// TwinCAT 3 PLC project TestIOC
// ProgramVersion: 3.1.4026.17
// libraries:
//   LCLS General, * (SLAC)
//   LCLS Vacuum, * (SLAC - LCLS)
//   lcls-twincat-common-components, * (SLAC)
//   lcls-twincat-math, * (SLAC - LCLS)
//   lcls-twincat-motion, * (SLAC)
//   lcls-twincat-optics, * (SLAC)
//   lcls-twincat-physics, * (SLAC)
//   LCLS_MotionAbstraction, * (SLAC)
//   LCLS_Tc_DevAbs, * (SLAC - LCLS)
//   PMPS, * (SLAC - LCLS)
//   Tc2_MC2, * (Beckhoff Automation GmbH)
//   Tc2_Standard, * (Beckhoff Automation GmbH)
//   Tc2_System, * (Beckhoff Automation GmbH)
//   Tc3_Module, * (Beckhoff Automation GmbH)
//   TcUnit, * (www.tcunit.org)
// project tree:
//   DUTs/ ENUM_Test.TcDUT, ST_NestedTypes01.TcDUT, ST_NestedTypes02.TcDUT, ST_NestedTypes03.TcDUT, ST_NestedTypes04.TcDUT, ST_NestedTypes05.TcDUT, ST_PytmcTypes.TcDUT
//   GVLs/ GVL.TcGVL
//   / PlcTask.TcTTO
//   POUs/ Main.TcPOU, F_UpdateArray.TcPOU
// real-time tasks:
//   TASK PlcTask: cycle T#10ms, priority 20, ADS port 350
// motion (NC):
//   TASK NC-Task 1 SAF: cycle T#2ms, priority 4, ADS port 501
//   TASK NC-Task 1 SVB: cycle T#10ms, priority 8, ADS port 511
//   AXIS Axis 1 (id 1)
//     OtherSettings: AllowMotionCmdToSlave=true
//     encoder EncType=1
//     drive DrvType=5
//       Analog: TorqueSetpointScale=10, ScaleFactorActTorque=0.1
//       TimeComp: TaskDelayCycles=1
//     controller CtrType=1
//       CtrPara: PriorControlFactor=1
//         Observer: BandWidth=20
//   AXIS Axis 2 (id 2)
//     OtherSettings: AllowMotionCmdToSlave=true
//     encoder EncType=1
//     drive DrvType=5
//       Analog: TorqueSetpointScale=10, ScaleFactorActTorque=0.1
//       TimeComp: TaskDelayCycles=1
//     controller CtrType=1
//       CtrPara: PriorControlFactor=1
//         Observer: BandWidth=20
//   AXIS Axis 3 (id 3)
//     OtherSettings: AllowMotionCmdToSlave=true
//     encoder EncType=1
//     drive DrvType=5
//       Analog: TorqueSetpointScale=10, ScaleFactorActTorque=0.1
//       TimeComp: TaskDelayCycles=1
//     controller CtrType=1
//       CtrPara: PriorControlFactor=1
//         Observer: BandWidth=20
//   AXIS Axis 4 (id 4)
//     OtherSettings: AllowMotionCmdToSlave=true
//     encoder EncType=1
//     drive DrvType=5
//       Analog: TorqueSetpointScale=10, ScaleFactorActTorque=0.1
//       TimeComp: TaskDelayCycles=1
//     controller CtrType=1
//       CtrPara: PriorControlFactor=1
//         Observer: BandWidth=20
//   AXIS Axis 5 (id 5)
//     OtherSettings: AllowMotionCmdToSlave=true
//     encoder EncType=1
//     drive DrvType=5
//       Analog: TorqueSetpointScale=10, ScaleFactorActTorque=0.1
//       TimeComp: TaskDelayCycles=1
//     controller CtrType=1
//       CtrPara: PriorControlFactor=1
//         Observer: BandWidth=20
//   AXIS Axis 6 (id 6)
//     OtherSettings: AllowMotionCmdToSlave=true
//     encoder EncType=1
//     drive DrvType=5
//       Analog: TorqueSetpointScale=10, ScaleFactorActTorque=0.1
//       TimeComp: TaskDelayCycles=1
//     controller CtrType=1
//       CtrPara: PriorControlFactor=1
//         Observer: BandWidth=20
//   AXIS Axis 7 (id 7)
//     OtherSettings: AllowMotionCmdToSlave=true
//     encoder EncType=1
//     drive DrvType=5
//       Analog: TorqueSetpointScale=10, ScaleFactorActTorque=0.1
//       TimeComp: TaskDelayCycles=1
//     controller CtrType=1
//       CtrPara: PriorControlFactor=1
//         Observer: BandWidth=20
//   AXIS Axis 8 (id 8)
//     OtherSettings: AllowMotionCmdToSlave=true
//     encoder EncType=1
//     drive DrvType=5
//       Analog: TorqueSetpointScale=10, ScaleFactorActTorque=0.1
//       TimeComp: TaskDelayCycles=1
//     controller CtrType=1
//       CtrPara: PriorControlFactor=1
//         Observer: BandWidth=20
//   AXIS Axis 9 (id 9)
//     OtherSettings: AllowMotionCmdToSlave=true
//     encoder EncType=1
//     drive DrvType=5
//       Analog: TorqueSetpointScale=10, ScaleFactorActTorque=0.1
//       TimeComp: TaskDelayCycles=1
//     controller CtrType=1
//       CtrPara: PriorControlFactor=1
//         Observer: BandWidth=20
//   AXIS Axis 10 (id 10)
//     OtherSettings: AllowMotionCmdToSlave=true
//     encoder EncType=1
//     drive DrvType=5
//       Analog: TorqueSetpointScale=10, ScaleFactorActTorque=0.1
//       TimeComp: TaskDelayCycles=1
//     controller CtrType=1
//       CtrPara: PriorControlFactor=1
//         Observer: BandWidth=20
//   AXIS Axis 11 (id 11)
//     OtherSettings: AllowMotionCmdToSlave=true
//     encoder EncType=1
//     drive DrvType=5
//       Analog: TorqueSetpointScale=10, ScaleFactorActTorque=0.1
//       TimeComp: TaskDelayCycles=1
//     controller CtrType=1
//       CtrPara: PriorControlFactor=1
//         Observer: BandWidth=20
//   AXIS Axis 12 (id 12)
//     OtherSettings: AllowMotionCmdToSlave=true
//     encoder EncType=1
//     drive DrvType=5
//       Analog: TorqueSetpointScale=10, ScaleFactorActTorque=0.1
//       TimeComp: TaskDelayCycles=1
//     controller CtrType=1
//       CtrPara: PriorControlFactor=1
//         Observer: BandWidth=20
//   AXIS Axis 13 (id 13)
//     OtherSettings: AllowMotionCmdToSlave=true
//     encoder EncType=1
//     drive DrvType=5
//       Analog: TorqueSetpointScale=10, ScaleFactorActTorque=0.1
//       TimeComp: TaskDelayCycles=1
//     controller CtrType=1
//       CtrPara: PriorControlFactor=1
//         Observer: BandWidth=20
//   AXIS Axis 14 (id 14)
//     OtherSettings: AllowMotionCmdToSlave=true
//     encoder EncType=1
//     drive DrvType=5
//       Analog: TorqueSetpointScale=10, ScaleFactorActTorque=0.1
//       TimeComp: TaskDelayCycles=1
//     controller CtrType=1
//       CtrPara: PriorControlFactor=1
//         Observer: BandWidth=20
//   AXIS Axis 15 (id 15)
//     OtherSettings: AllowMotionCmdToSlave=true
//     encoder EncType=1
//     drive DrvType=5
//       Analog: TorqueSetpointScale=10, ScaleFactorActTorque=0.1
//       TimeComp: TaskDelayCycles=1
//     controller CtrType=1
//       CtrPara: PriorControlFactor=1
//         Observer: BandWidth=20
//   AXIS Axis 16 (id 16)
//     OtherSettings: AllowMotionCmdToSlave=true
//     encoder EncType=1
//     drive DrvType=5
//       Analog: TorqueSetpointScale=10, ScaleFactorActTorque=0.1
//       TimeComp: TaskDelayCycles=1
//     controller CtrType=1
//       CtrPara: PriorControlFactor=1
//         Observer: BandWidth=20
//   AXIS Axis 17 (id 17)
//     OtherSettings: AllowMotionCmdToSlave=true
//     encoder EncType=1
//     drive DrvType=5
//       Analog: TorqueSetpointScale=10, ScaleFactorActTorque=0.1
//       TimeComp: TaskDelayCycles=1
//     controller CtrType=1
//       CtrPara: PriorControlFactor=1
//         Observer: BandWidth=20
//   AXIS Axis 18 (id 18)
//     OtherSettings: AllowMotionCmdToSlave=true
//     encoder EncType=1
//     drive DrvType=5
//       Analog: TorqueSetpointScale=10, ScaleFactorActTorque=0.1
//       TimeComp: TaskDelayCycles=1
//     controller CtrType=1
//       CtrPara: PriorControlFactor=1
//         Observer: BandWidth=20
//   AXIS Axis 19 (id 19)
//     OtherSettings: AllowMotionCmdToSlave=true
//     encoder EncType=1
//     drive DrvType=5
//       Analog: TorqueSetpointScale=10, ScaleFactorActTorque=0.1
//       TimeComp: TaskDelayCycles=1
//     controller CtrType=1
//       CtrPara: PriorControlFactor=1
//         Observer: BandWidth=20
//   AXIS Axis 20 (id 20)
//     OtherSettings: AllowMotionCmdToSlave=true
//     encoder EncType=1
//     drive DrvType=5
//       Analog: TorqueSetpointScale=10, ScaleFactorActTorque=0.1
//       TimeComp: TaskDelayCycles=1
//     controller CtrType=1
//       CtrPara: PriorControlFactor=1
//         Observer: BandWidth=20
//   AXIS Axis 21 (id 21)
//     OtherSettings: AllowMotionCmdToSlave=true
//     encoder EncType=1
//     drive DrvType=5
//       Analog: TorqueSetpointScale=10, ScaleFactorActTorque=0.1
//       TimeComp: TaskDelayCycles=1
//     controller CtrType=1
//       CtrPara: PriorControlFactor=1
//         Observer: BandWidth=20
//   AXIS Axis 22 (id 22)
//     OtherSettings: AllowMotionCmdToSlave=true
//     encoder EncType=1
//     drive DrvType=5
//       Analog: TorqueSetpointScale=10, ScaleFactorActTorque=0.1
//       TimeComp: TaskDelayCycles=1
//     controller CtrType=1
//       CtrPara: PriorControlFactor=1
//         Observer: BandWidth=20
//   AXIS Axis 23 (id 23)
//     OtherSettings: AllowMotionCmdToSlave=true
//     encoder EncType=1
//     drive DrvType=5
//       Analog: TorqueSetpointScale=10, ScaleFactorActTorque=0.1
//       TimeComp: TaskDelayCycles=1
//     controller CtrType=1
//       CtrPara: PriorControlFactor=1
//         Observer: BandWidth=20
//   AXIS Axis 24 (id 24)
//     OtherSettings: AllowMotionCmdToSlave=true
//     encoder EncType=1
//     drive DrvType=5
//       Analog: TorqueSetpointScale=10, ScaleFactorActTorque=0.1
//       TimeComp: TaskDelayCycles=1
//     controller CtrType=1
//       CtrPara: PriorControlFactor=1
//         Observer: BandWidth=20
//   AXIS Axis 25 (id 25)
//     OtherSettings: AllowMotionCmdToSlave=true
//     encoder EncType=1
//     drive DrvType=5
//       Analog: TorqueSetpointScale=10, ScaleFactorActTorque=0.1
//       TimeComp: TaskDelayCycles=1
//     controller CtrType=1
//       CtrPara: PriorControlFactor=1
//         Observer: BandWidth=20
//   AXIS Axis 26 (id 26)
//     OtherSettings: AllowMotionCmdToSlave=true
//     encoder EncType=1
//     drive DrvType=5
//       Analog: TorqueSetpointScale=10, ScaleFactorActTorque=0.1
//       TimeComp: TaskDelayCycles=1
//     controller CtrType=1
//       CtrPara: PriorControlFactor=1
//         Observer: BandWidth=20
//   AXIS Axis 27 (id 27)
//     OtherSettings: AllowMotionCmdToSlave=true
//     encoder EncType=1
//     drive DrvType=5
//       Analog: TorqueSetpointScale=10, ScaleFactorActTorque=0.1
//       TimeComp: TaskDelayCycles=1
//     controller CtrType=1
//       CtrPara: PriorControlFactor=1
//         Observer: BandWidth=20
//   AXIS Axis 28 (id 28)
//     OtherSettings: AllowMotionCmdToSlave=true
//     encoder EncType=1
//     drive DrvType=5
//       Analog: TorqueSetpointScale=10, ScaleFactorActTorque=0.1
//       TimeComp: TaskDelayCycles=1
//     controller CtrType=1
//       CtrPara: PriorControlFactor=1
//         Observer: BandWidth=20
//   AXIS Axis 29 (id 29)
//     OtherSettings: AllowMotionCmdToSlave=true
//     encoder EncType=1
//     drive DrvType=5
//       Analog: TorqueSetpointScale=10, ScaleFactorActTorque=0.1
//       TimeComp: TaskDelayCycles=1
//     controller CtrType=1
//       CtrPara: PriorControlFactor=1
//         Observer: BandWidth=20
//   AXIS Axis 30 (id 30)
//     OtherSettings: AllowMotionCmdToSlave=true
//     encoder EncType=1
//     drive DrvType=5
//       Analog: TorqueSetpointScale=10, ScaleFactorActTorque=0.1
//       TimeComp: TaskDelayCycles=1
//     controller CtrType=1
//       CtrPara: PriorControlFactor=1
//         Observer: BandWidth=20
//   AXIS Axis 31 (id 31)
//     OtherSettings: AllowMotionCmdToSlave=true
//     encoder EncType=1
//     drive DrvType=5
//       Analog: TorqueSetpointScale=10, ScaleFactorActTorque=0.1
//       TimeComp: TaskDelayCycles=1
//     controller CtrType=1
//       CtrPara: PriorControlFactor=1
//         Observer: BandWidth=20
//   AXIS Axis 32 (id 32)
//     OtherSettings: AllowMotionCmdToSlave=true
//     encoder EncType=1
//     drive DrvType=5
//       Analog: TorqueSetpointScale=10, ScaleFactorActTorque=0.1
//       TimeComp: TaskDelayCycles=1
//     controller CtrType=1
//       CtrPara: PriorControlFactor=1
//         Observer: BandWidth=20
//   AXIS Axis 33 (id 33)
//     OtherSettings: AllowMotionCmdToSlave=true
//     encoder EncType=1
//     drive DrvType=5
//       Analog: TorqueSetpointScale=10, ScaleFactorActTorque=0.1
//       TimeComp: TaskDelayCycles=1
//     controller CtrType=1
//       CtrPara: PriorControlFactor=1
//         Observer: BandWidth=20
//   AXIS Axis 34 (id 34)
//     OtherSettings: AllowMotionCmdToSlave=true
//     encoder EncType=1
//     drive DrvType=5
//       Analog: TorqueSetpointScale=10, ScaleFactorActTorque=0.1
//       TimeComp: TaskDelayCycles=1
//     controller CtrType=1
//       CtrPara: PriorControlFactor=1
//         Observer: BandWidth=20
//   AXIS Axis 35 (id 35)
//     OtherSettings: AllowMotionCmdToSlave=true
//     encoder EncType=1
//     drive DrvType=5
//       Analog: TorqueSetpointScale=10, ScaleFactorActTorque=0.1
//       TimeComp: TaskDelayCycles=1
//     controller CtrType=1
//       CtrPara: PriorControlFactor=1
//         Observer: BandWidth=20
//   AXIS Axis 36 (id 36)
//     OtherSettings: AllowMotionCmdToSlave=true
//     encoder EncType=1
//     drive DrvType=5
//       Analog: TorqueSetpointScale=10, ScaleFactorActTorque=0.1
//       TimeComp: TaskDelayCycles=1
//     controller CtrType=1
//       CtrPara: PriorControlFactor=1
//         Observer: BandWidth=20
//   AXIS Axis 37 (id 37)
//     OtherSettings: AllowMotionCmdToSlave=true
//     encoder EncType=1
//     drive DrvType=5
//       Analog: TorqueSetpointScale=10, ScaleFactorActTorque=0.1
//       TimeComp: TaskDelayCycles=1
//     controller CtrType=1
//       CtrPara: PriorControlFactor=1
//         Observer: BandWidth=20
//   AXIS Axis 38 (id 38)
//     OtherSettings: AllowMotionCmdToSlave=true
//     encoder EncType=1
//     drive DrvType=5
//       Analog: TorqueSetpointScale=10, ScaleFactorActTorque=0.1
//       TimeComp: TaskDelayCycles=1
//     controller CtrType=1
//       CtrPara: PriorControlFactor=1
//         Observer: BandWidth=20
//   AXIS Axis 39 (id 39)
//     OtherSettings: AllowMotionCmdToSlave=true
//     encoder EncType=1
//     drive DrvType=5
//       Analog: TorqueSetpointScale=10, ScaleFactorActTorque=0.1
//       TimeComp: TaskDelayCycles=1
//     controller CtrType=1
//       CtrPara: PriorControlFactor=1
//         Observer: BandWidth=20
//   AXIS Axis 40 (id 40)
//     OtherSettings: AllowMotionCmdToSlave=true
//     encoder EncType=1
//     drive DrvType=5
//       Analog: TorqueSetpointScale=10, ScaleFactorActTorque=0.1
//       TimeComp: TaskDelayCycles=1
//     controller CtrType=1
//       CtrPara: PriorControlFactor=1
//         Observer: BandWidth=20
//   AXIS Axis 41 (id 41)
//     OtherSettings: AllowMotionCmdToSlave=true
//     encoder EncType=1
//     drive DrvType=5
//       Analog: TorqueSetpointScale=10, ScaleFactorActTorque=0.1
//       TimeComp: TaskDelayCycles=1
//     controller CtrType=1
//       CtrPara: PriorControlFactor=1
//         Observer: BandWidth=20
//   AXIS Axis 42 (id 42)
//     OtherSettings: AllowMotionCmdToSlave=true
//     encoder EncType=1
//     drive DrvType=5
//       Analog: TorqueSetpointScale=10, ScaleFactorActTorque=0.1
//       TimeComp: TaskDelayCycles=1
//     controller CtrType=1
//       CtrPara: PriorControlFactor=1
//         Observer: BandWidth=20
//   AXIS Axis 43 (id 43)
//     OtherSettings: AllowMotionCmdToSlave=true
//     encoder EncType=1
//     drive DrvType=5
//       Analog: TorqueSetpointScale=10, ScaleFactorActTorque=0.1
//       TimeComp: TaskDelayCycles=1
//     controller CtrType=1
//       CtrPara: PriorControlFactor=1
//         Observer: BandWidth=20
//   AXIS Axis 44 (id 44)
//     OtherSettings: AllowMotionCmdToSlave=true
//     encoder EncType=1
//     drive DrvType=5
//       Analog: TorqueSetpointScale=10, ScaleFactorActTorque=0.1
//       TimeComp: TaskDelayCycles=1
//     controller CtrType=1
//       CtrPara: PriorControlFactor=1
//         Observer: BandWidth=20
//   AXIS Axis 45 (id 45)
//     OtherSettings: AllowMotionCmdToSlave=true
//     encoder EncType=1
//     drive DrvType=5
//       Analog: TorqueSetpointScale=10, ScaleFactorActTorque=0.1
//       TimeComp: TaskDelayCycles=1
//     controller CtrType=1
//       CtrPara: PriorControlFactor=1
//         Observer: BandWidth=20
//   AXIS Axis 46 (id 46)
//     OtherSettings: AllowMotionCmdToSlave=true
//     encoder EncType=1
//     drive DrvType=5
//       Analog: TorqueSetpointScale=10, ScaleFactorActTorque=0.1
//       TimeComp: TaskDelayCycles=1
//     controller CtrType=1
//       CtrPara: PriorControlFactor=1
//         Observer: BandWidth=20
//   AXIS Axis 47 (id 47)
//     OtherSettings: AllowMotionCmdToSlave=true
//     encoder EncType=1
//     drive DrvType=5
//       Analog: TorqueSetpointScale=10, ScaleFactorActTorque=0.1
//       TimeComp: TaskDelayCycles=1
//     controller CtrType=1
//       CtrPara: PriorControlFactor=1
//         Observer: BandWidth=20
//   AXIS Axis 48 (id 48)
//     OtherSettings: AllowMotionCmdToSlave=true
//     encoder EncType=1
//     drive DrvType=5
//       Analog: TorqueSetpointScale=10, ScaleFactorActTorque=0.1
//       TimeComp: TaskDelayCycles=1
//     controller CtrType=1
//       CtrPara: PriorControlFactor=1
//         Observer: BandWidth=20
//   AXIS Axis 49 (id 49)
//     OtherSettings: AllowMotionCmdToSlave=true
//     encoder EncType=1
//     drive DrvType=5
//       Analog: TorqueSetpointScale=10, ScaleFactorActTorque=0.1
//       TimeComp: TaskDelayCycles=1
//     controller CtrType=1
//       CtrPara: PriorControlFactor=1
//         Observer: BandWidth=20
//   AXIS Axis 50 (id 50)
//     OtherSettings: AllowMotionCmdToSlave=true
//     encoder EncType=1
//     drive DrvType=5
//       Analog: TorqueSetpointScale=10, ScaleFactorActTorque=0.1
//       TimeComp: TaskDelayCycles=1
//     controller CtrType=1
//       CtrPara: PriorControlFactor=1
//         Observer: BandWidth=20
//   AXIS Axis 51 (id 51)
//     OtherSettings: AllowMotionCmdToSlave=true
//     encoder EncType=1
//     drive DrvType=5
//       Analog: TorqueSetpointScale=10, ScaleFactorActTorque=0.1
//       TimeComp: TaskDelayCycles=1
//     controller CtrType=1
//       CtrPara: PriorControlFactor=1
//         Observer: BandWidth=20
//   AXIS Axis 52 (id 52)
//     OtherSettings: AllowMotionCmdToSlave=true
//     encoder EncType=1
//     drive DrvType=5
//       Analog: TorqueSetpointScale=10, ScaleFactorActTorque=0.1
//       TimeComp: TaskDelayCycles=1
//     controller CtrType=1
//       CtrPara: PriorControlFactor=1
//         Observer: BandWidth=20
// variable links:
//   (this object) <-> NC-Task 1 SAF/Axes/Axis 1
//     PlcTask Inputs/Main.M1.Axis.NcToPlc <-> Outputs/ToPlc
//     PlcTask Outputs/Main.M1.Axis.PlcToNc <-> Inputs/FromPlc
//   (this object) <-> NC-Task 1 SAF/Axes/Axis 10
//     PlcTask Inputs/Main.aAxisRef[8].NcToPlc <-> Outputs/ToPlc
//     PlcTask Outputs/Main.aAxisRef[8].PlcToNc <-> Inputs/FromPlc
//   (this object) <-> NC-Task 1 SAF/Axes/Axis 11
//     PlcTask Inputs/Main.aAxisRef[9].NcToPlc <-> Outputs/ToPlc
//     PlcTask Outputs/Main.aAxisRef[9].PlcToNc <-> Inputs/FromPlc
//   (this object) <-> NC-Task 1 SAF/Axes/Axis 12
//     PlcTask Inputs/Main.aAxisRef[10].NcToPlc <-> Outputs/ToPlc
//     PlcTask Outputs/Main.aAxisRef[10].PlcToNc <-> Inputs/FromPlc
//   (this object) <-> NC-Task 1 SAF/Axes/Axis 13
//     PlcTask Inputs/Main.aAxisRef[11].NcToPlc <-> Outputs/ToPlc
//     PlcTask Outputs/Main.aAxisRef[11].PlcToNc <-> Inputs/FromPlc
//   (this object) <-> NC-Task 1 SAF/Axes/Axis 14
//     PlcTask Inputs/Main.aAxisRef[12].NcToPlc <-> Outputs/ToPlc
//     PlcTask Outputs/Main.aAxisRef[12].PlcToNc <-> Inputs/FromPlc
//   (this object) <-> NC-Task 1 SAF/Axes/Axis 15
//     PlcTask Inputs/Main.aAxisRef[13].NcToPlc <-> Outputs/ToPlc
//     PlcTask Outputs/Main.aAxisRef[13].PlcToNc <-> Inputs/FromPlc
//   (this object) <-> NC-Task 1 SAF/Axes/Axis 16
//     PlcTask Inputs/Main.aAxisRef[14].NcToPlc <-> Outputs/ToPlc
//     PlcTask Outputs/Main.aAxisRef[14].PlcToNc <-> Inputs/FromPlc
//   (this object) <-> NC-Task 1 SAF/Axes/Axis 17
//     PlcTask Inputs/Main.aAxisRef[15].NcToPlc <-> Outputs/ToPlc
//     PlcTask Outputs/Main.aAxisRef[15].PlcToNc <-> Inputs/FromPlc
//   (this object) <-> NC-Task 1 SAF/Axes/Axis 18
//     PlcTask Inputs/Main.aAxisRef[16].NcToPlc <-> Outputs/ToPlc
//     PlcTask Outputs/Main.aAxisRef[16].PlcToNc <-> Inputs/FromPlc
//   (this object) <-> NC-Task 1 SAF/Axes/Axis 19
//     PlcTask Inputs/Main.aAxisRef[17].NcToPlc <-> Outputs/ToPlc
//     PlcTask Outputs/Main.aAxisRef[17].PlcToNc <-> Inputs/FromPlc
//   (this object) <-> NC-Task 1 SAF/Axes/Axis 2
//     PlcTask Inputs/Main.M2.Axis.NcToPlc <-> Outputs/ToPlc
//     PlcTask Outputs/Main.M2.Axis.PlcToNc <-> Inputs/FromPlc
//   (this object) <-> NC-Task 1 SAF/Axes/Axis 20
//     PlcTask Inputs/Main.aAxisRef[18].NcToPlc <-> Outputs/ToPlc
//     PlcTask Outputs/Main.aAxisRef[18].PlcToNc <-> Inputs/FromPlc
//   (this object) <-> NC-Task 1 SAF/Axes/Axis 21
//     PlcTask Inputs/Main.aAxisRef[19].NcToPlc <-> Outputs/ToPlc
//     PlcTask Outputs/Main.aAxisRef[19].PlcToNc <-> Inputs/FromPlc
//   (this object) <-> NC-Task 1 SAF/Axes/Axis 22
//     PlcTask Inputs/Main.aAxisRef[20].NcToPlc <-> Outputs/ToPlc
//     PlcTask Outputs/Main.aAxisRef[20].PlcToNc <-> Inputs/FromPlc
//   (this object) <-> NC-Task 1 SAF/Axes/Axis 23
//     PlcTask Inputs/Main.aAxisRef[21].NcToPlc <-> Outputs/ToPlc
//     PlcTask Outputs/Main.aAxisRef[21].PlcToNc <-> Inputs/FromPlc
//   (this object) <-> NC-Task 1 SAF/Axes/Axis 24
//     PlcTask Inputs/Main.aAxisRef[22].NcToPlc <-> Outputs/ToPlc
//     PlcTask Outputs/Main.aAxisRef[22].PlcToNc <-> Inputs/FromPlc
//   (this object) <-> NC-Task 1 SAF/Axes/Axis 25
//     PlcTask Inputs/Main.aAxisRef[23].NcToPlc <-> Outputs/ToPlc
//     PlcTask Outputs/Main.aAxisRef[23].PlcToNc <-> Inputs/FromPlc
//   (this object) <-> NC-Task 1 SAF/Axes/Axis 26
//     PlcTask Inputs/Main.aAxisRef[24].NcToPlc <-> Outputs/ToPlc
//     PlcTask Outputs/Main.aAxisRef[24].PlcToNc <-> Inputs/FromPlc
//   (this object) <-> NC-Task 1 SAF/Axes/Axis 27
//     PlcTask Inputs/Main.aAxisRef[25].NcToPlc <-> Outputs/ToPlc
//     PlcTask Outputs/Main.aAxisRef[25].PlcToNc <-> Inputs/FromPlc
//   (this object) <-> NC-Task 1 SAF/Axes/Axis 28
//     PlcTask Inputs/Main.aAxisRef[26].NcToPlc <-> Outputs/ToPlc
//     PlcTask Outputs/Main.aAxisRef[26].PlcToNc <-> Inputs/FromPlc
//   (this object) <-> NC-Task 1 SAF/Axes/Axis 29
//     PlcTask Inputs/Main.aAxisRef[27].NcToPlc <-> Outputs/ToPlc
//     PlcTask Outputs/Main.aAxisRef[27].PlcToNc <-> Inputs/FromPlc
//   (this object) <-> NC-Task 1 SAF/Axes/Axis 3
//     PlcTask Inputs/Main.aAxisRef[1].NcToPlc <-> Outputs/ToPlc
//     PlcTask Outputs/Main.aAxisRef[1].PlcToNc <-> Inputs/FromPlc
//   (this object) <-> NC-Task 1 SAF/Axes/Axis 30
//     PlcTask Inputs/Main.aAxisRef[28].NcToPlc <-> Outputs/ToPlc
//     PlcTask Outputs/Main.aAxisRef[28].PlcToNc <-> Inputs/FromPlc
//   (this object) <-> NC-Task 1 SAF/Axes/Axis 31
//     PlcTask Inputs/Main.aAxisRef[29].NcToPlc <-> Outputs/ToPlc
//     PlcTask Outputs/Main.aAxisRef[29].PlcToNc <-> Inputs/FromPlc
//   (this object) <-> NC-Task 1 SAF/Axes/Axis 32
//     PlcTask Inputs/Main.aAxisRef[30].NcToPlc <-> Outputs/ToPlc
//     PlcTask Outputs/Main.aAxisRef[30].PlcToNc <-> Inputs/FromPlc
//   (this object) <-> NC-Task 1 SAF/Axes/Axis 33
//     PlcTask Inputs/Main.aAxisRef[31].NcToPlc <-> Outputs/ToPlc
//     PlcTask Outputs/Main.aAxisRef[31].PlcToNc <-> Inputs/FromPlc
//   (this object) <-> NC-Task 1 SAF/Axes/Axis 34
//     PlcTask Inputs/Main.aAxisRef[32].NcToPlc <-> Outputs/ToPlc
//     PlcTask Outputs/Main.aAxisRef[32].PlcToNc <-> Inputs/FromPlc
//   (this object) <-> NC-Task 1 SAF/Axes/Axis 35
//     PlcTask Inputs/Main.aAxisRef[33].NcToPlc <-> Outputs/ToPlc
//     PlcTask Outputs/Main.aAxisRef[33].PlcToNc <-> Inputs/FromPlc
//   (this object) <-> NC-Task 1 SAF/Axes/Axis 36
//     PlcTask Inputs/Main.aAxisRef[34].NcToPlc <-> Outputs/ToPlc
//     PlcTask Outputs/Main.aAxisRef[34].PlcToNc <-> Inputs/FromPlc
//   (this object) <-> NC-Task 1 SAF/Axes/Axis 37
//     PlcTask Inputs/Main.aAxisRef[35].NcToPlc <-> Outputs/ToPlc
//     PlcTask Outputs/Main.aAxisRef[35].PlcToNc <-> Inputs/FromPlc
//   (this object) <-> NC-Task 1 SAF/Axes/Axis 38
//     PlcTask Inputs/Main.aAxisRef[36].NcToPlc <-> Outputs/ToPlc
//     PlcTask Outputs/Main.aAxisRef[36].PlcToNc <-> Inputs/FromPlc
//   (this object) <-> NC-Task 1 SAF/Axes/Axis 39
//     PlcTask Inputs/Main.aAxisRef[37].NcToPlc <-> Outputs/ToPlc
//     PlcTask Outputs/Main.aAxisRef[37].PlcToNc <-> Inputs/FromPlc
//   (this object) <-> NC-Task 1 SAF/Axes/Axis 4
//     PlcTask Inputs/Main.aAxisRef[2].NcToPlc <-> Outputs/ToPlc
//     PlcTask Outputs/Main.aAxisRef[2].PlcToNc <-> Inputs/FromPlc
//   (this object) <-> NC-Task 1 SAF/Axes/Axis 40
//     PlcTask Inputs/Main.aAxisRef[38].NcToPlc <-> Outputs/ToPlc
//     PlcTask Outputs/Main.aAxisRef[38].PlcToNc <-> Inputs/FromPlc
//   (this object) <-> NC-Task 1 SAF/Axes/Axis 41
//     PlcTask Inputs/Main.aAxisRef[39].NcToPlc <-> Outputs/ToPlc
//     PlcTask Outputs/Main.aAxisRef[39].PlcToNc <-> Inputs/FromPlc
//   (this object) <-> NC-Task 1 SAF/Axes/Axis 42
//     PlcTask Inputs/Main.aAxisRef[40].NcToPlc <-> Outputs/ToPlc
//     PlcTask Outputs/Main.aAxisRef[40].PlcToNc <-> Inputs/FromPlc
//   (this object) <-> NC-Task 1 SAF/Axes/Axis 43
//     PlcTask Inputs/Main.aAxisRef[41].NcToPlc <-> Outputs/ToPlc
//     PlcTask Outputs/Main.aAxisRef[41].PlcToNc <-> Inputs/FromPlc
//   (this object) <-> NC-Task 1 SAF/Axes/Axis 44
//     PlcTask Inputs/Main.aAxisRef[42].NcToPlc <-> Outputs/ToPlc
//     PlcTask Outputs/Main.aAxisRef[42].PlcToNc <-> Inputs/FromPlc
//   (this object) <-> NC-Task 1 SAF/Axes/Axis 45
//     PlcTask Inputs/Main.aAxisRef[43].NcToPlc <-> Outputs/ToPlc
//     PlcTask Outputs/Main.aAxisRef[43].PlcToNc <-> Inputs/FromPlc
//   (this object) <-> NC-Task 1 SAF/Axes/Axis 46
//     PlcTask Inputs/Main.aAxisRef[44].NcToPlc <-> Outputs/ToPlc
//     PlcTask Outputs/Main.aAxisRef[44].PlcToNc <-> Inputs/FromPlc
//   (this object) <-> NC-Task 1 SAF/Axes/Axis 47
//     PlcTask Inputs/Main.aAxisRef[45].NcToPlc <-> Outputs/ToPlc
//     PlcTask Outputs/Main.aAxisRef[45].PlcToNc <-> Inputs/FromPlc
//   (this object) <-> NC-Task 1 SAF/Axes/Axis 48
//     PlcTask Inputs/Main.aAxisRef[46].NcToPlc <-> Outputs/ToPlc
//     PlcTask Outputs/Main.aAxisRef[46].PlcToNc <-> Inputs/FromPlc
//   (this object) <-> NC-Task 1 SAF/Axes/Axis 49
//     PlcTask Inputs/Main.aAxisRef[47].NcToPlc <-> Outputs/ToPlc
//     PlcTask Outputs/Main.aAxisRef[47].PlcToNc <-> Inputs/FromPlc
//   (this object) <-> NC-Task 1 SAF/Axes/Axis 5
//     PlcTask Inputs/Main.aAxisRef[3].NcToPlc <-> Outputs/ToPlc
//     PlcTask Outputs/Main.aAxisRef[3].PlcToNc <-> Inputs/FromPlc
//   (this object) <-> NC-Task 1 SAF/Axes/Axis 50
//     PlcTask Inputs/Main.aAxisRef[48].NcToPlc <-> Outputs/ToPlc
//     PlcTask Outputs/Main.aAxisRef[48].PlcToNc <-> Inputs/FromPlc
//   (this object) <-> NC-Task 1 SAF/Axes/Axis 51
//     PlcTask Inputs/Main.aAxisRef[49].NcToPlc <-> Outputs/ToPlc
//     PlcTask Outputs/Main.aAxisRef[49].PlcToNc <-> Inputs/FromPlc
//   (this object) <-> NC-Task 1 SAF/Axes/Axis 52
//     PlcTask Inputs/Main.aAxisRef[50].NcToPlc <-> Outputs/ToPlc
//     PlcTask Outputs/Main.aAxisRef[50].PlcToNc <-> Inputs/FromPlc
//   (this object) <-> NC-Task 1 SAF/Axes/Axis 6
//     PlcTask Inputs/Main.aAxisRef[4].NcToPlc <-> Outputs/ToPlc
//     PlcTask Outputs/Main.aAxisRef[4].PlcToNc <-> Inputs/FromPlc
//   (this object) <-> NC-Task 1 SAF/Axes/Axis 7
//     PlcTask Inputs/Main.aAxisRef[5].NcToPlc <-> Outputs/ToPlc
//     PlcTask Outputs/Main.aAxisRef[5].PlcToNc <-> Inputs/FromPlc
//   (this object) <-> NC-Task 1 SAF/Axes/Axis 8
//     PlcTask Inputs/Main.aAxisRef[6].NcToPlc <-> Outputs/ToPlc
//     PlcTask Outputs/Main.aAxisRef[6].PlcToNc <-> Inputs/FromPlc
//   (this object) <-> NC-Task 1 SAF/Axes/Axis 9
//     PlcTask Inputs/Main.aAxisRef[7].NcToPlc <-> Outputs/ToPlc
//     PlcTask Outputs/Main.aAxisRef[7].PlcToNc <-> Inputs/FromPlc

CONFIGURATION TestIOC
    RESOURCE PLC ON TwinCAT3
        TASK PlcTask(INTERVAL := T#10ms, PRIORITY := 20);
        PROGRAM Main WITH PlcTask : Main;
    END_RESOURCE
END_CONFIGURATION

// ---- DUTs/ENUM_Test.TcDUT
{attribute 'qualified_only'}
{attribute 'strict'}
TYPE ENUM_Test :
(
    zero := 0,
    one := 1,
    two := 2,
    three := 3,
    four := 4,
    five := 5,
    six := 6,
    seven := 7
);
END_TYPE

// ---- DUTs/ST_NestedTypes01.TcDUT

TYPE ST_NestedTypes01 :
STRUCT
	stPytmcTypes : ST_PytmcTypes;
	stNestedTypes : ST_NestedTypes02;
END_STRUCT
END_TYPE

// ---- DUTs/ST_NestedTypes02.TcDUT

TYPE ST_NestedTypes02 :
STRUCT
	stPytmcTypes : ST_PytmcTypes;
	stNestedTypes : ST_NestedTypes03;
END_STRUCT
END_TYPE

// ---- DUTs/ST_NestedTypes03.TcDUT

TYPE ST_NestedTypes03 :
STRUCT
	stPytmcTypes : ST_PytmcTypes;
	stNestedTypes : ST_NestedTypes04;
END_STRUCT
END_TYPE

// ---- DUTs/ST_NestedTypes04.TcDUT

TYPE ST_NestedTypes04 :
STRUCT
	stPytmcTypes : ST_PytmcTypes;
	stNestedTypes : ST_NestedTypes05;
END_STRUCT
END_TYPE

// ---- DUTs/ST_NestedTypes05.TcDUT

TYPE ST_NestedTypes05 :
STRUCT
	stPytmcTypes : ST_PytmcTypes;
END_STRUCT
END_TYPE

// ---- DUTs/ST_PytmcTypes.TcDUT

TYPE ST_PytmcTypes :
STRUCT
    {attribute 'pytmc' := 'pv: BOOL'}
    bBool: BOOL;
    {attribute 'pytmc' := 'pv: ARRAYBOOL'}
    arrBool: ARRAY[0..GVL.nPytmcTypesArrayLength] OF BOOL;
    {attribute 'pytmc' := 'pv: BYTE'}
    iByte: BYTE;
    {attribute 'pytmc' := 'pv: SINT'}
    iSint: SINT;
    {attribute 'pytmc' := 'pv: USINT'}
    iUsint: USINT;
    {attribute 'pytmc' := 'pv: WORD'}
    iWord: WORD;
    {attribute 'pytmc' := 'pv: INT'}
    iInt: INT;
    {attribute 'pytmc' := 'pv: ARRAYINT'}
    arrInt: ARRAY[0..GVL.nPytmcTypesArrayLength] OF INT;
    {attribute 'pytmc' := 'pv: UINT'}
    iUint: UINT;
    {attribute 'pytmc' := 'pv: ENUM'}
    eEnum: ENUM_Test;
    {attribute 'pytmc' := 'pv: ARRAYENUM'}
    arrUEnum: ARRAY[0..GVL.nPytmcTypesArrayLength] OF ENUM_Test;
    {attribute 'pytmc' := 'pv: DWORD'}
    iDword: DWORD;
    {attribute 'pytmc' := 'pv: DINT'}
    iDint: DINT;
    {attribute 'pytmc' := 'pv: ARRAYDINT'}
    arrDint: ARRAY[0..GVL.nPytmcTypesArrayLength] OF DINT;
    {attribute 'pytmc' := 'pv: UDINT'}
    iUdint: UDINT;
    {attribute 'pytmc' := 'pv: REAL'}
    fReal: REAL;
    {attribute 'pytmc' := 'pv: ARRAYREAL'}
    arrReal: ARRAY[0..GVL.nPytmcTypesArrayLength] OF REAL;
    {attribute 'pytmc' := 'pv: LREAL'}
    fLreal: LREAL;
    {attribute 'pytmc' := 'pv: ARRAYLREAL'}
    arrLreal: ARRAY[0..GVL.nPytmcTypesArrayLength] OF LREAL;
    {attribute 'pytmc' := 'pv: STRING'}
    sString: STRING;
    {attribute 'pytmc' := 'pv: MAXSTRING'}
    sMaxString: T_MaxString;
END_STRUCT
END_TYPE

// ---- GVLs/GVL.TcGVL

{attribute 'qualified_only'}
VAR_GLOBAL CONSTANT
	nPytmcTypesArrayLength : UINT := 99;
END_VAR

// ---- POUs/Main.TcPOU
PROGRAM Main
VAR CONSTANT
	nInArray : UINT := 250;
	nMotAbsAxes : UINT := 50;
END_VAR
VAR
	{attribute 'pytmc' := 'pv: @(PREFIX)M1'}
	{attribute 'TcNcAxis' := '.Axis := Axis 1'}
    M1: ST_MotionStage;
    {attribute 'pytmc' := 'pv: @(PREFIX)M2'}
	{attribute 'TcNcAxis' := '.Axis := Axis 2'}
    M2: ST_MotionStage;

    fbMotion01: FB_MotionStageSim;
    fbMotion02: FB_MotionStageSim;
	
	fbPersistentDataStorage: LCLS_Tc_DevAbs.FB_PersistentDataStorage;
	{attribute 'TcNcAxis' := '
		[1]  := Axis 3;
		[2]  := Axis 4;
		[3]  := Axis 5;
		[4]  := Axis 6;
		[5]  := Axis 7;
		[6]  := Axis 8;
		[7]  := Axis 9;
		[8]  := Axis 10;
		[9]  := Axis 11;
		[10] := Axis 12;
		[11] := Axis 13;
		[12] := Axis 14;
		[13] := Axis 15;
		[14] := Axis 16;
		[15] := Axis 17;
		[16] := Axis 18;
		[17] := Axis 19;
		[18] := Axis 20;
		[19] := Axis 21;
		[20] := Axis 22;
		[21] := Axis 23;
		[22] := Axis 24;
		[23] := Axis 25;
		[24] := Axis 26;
		[25] := Axis 27;
		[26] := Axis 28;
		[27] := Axis 29;
		[28] := Axis 30;
		[29] := Axis 31;
		[30] := Axis 32;
		[31] := Axis 33;
		[32] := Axis 34;
		[33] := Axis 35;
		[34] := Axis 36;
		[35] := Axis 37;
		[36] := Axis 38;
		[37] := Axis 39;
		[38] := Axis 40;
		[39] := Axis 41;
		[40] := Axis 42;
		[41] := Axis 43;
		[42] := Axis 44;
		[43] := Axis 45;
		[44] := Axis 46;
		[45] := Axis 47;
		[46] := Axis 48;
		[47] := Axis 49;
		[48] := Axis 50;
		[49] := Axis 51;
		[50] := Axis 52
	'}
	aAxisRef : ARRAY[1..nMotAbsAxes] OF AXIS_REF;
	{attribute 'pytmc' := 'pv: @(PREFIX)MOTABS'}
	fbMotionArr: ARRAY[1..nMotAbsAxes] OF FB_MotionStageNC[
		(AxisRef := aAxisRef[1],  iPersistentDataStorage := fbPersistentDataStorage, sName := 'Axis_03'),
		(AxisRef := aAxisRef[2],  iPersistentDataStorage := fbPersistentDataStorage, sName := 'Axis_02'),
		(AxisRef := aAxisRef[3],  iPersistentDataStorage := fbPersistentDataStorage, sName := 'Axis_03'),
		(AxisRef := aAxisRef[4],  iPersistentDataStorage := fbPersistentDataStorage, sName := 'Axis_04'),
		(AxisRef := aAxisRef[5],  iPersistentDataStorage := fbPersistentDataStorage, sName := 'Axis_05'),
		(AxisRef := aAxisRef[6],  iPersistentDataStorage := fbPersistentDataStorage, sName := 'Axis_06'),
		(AxisRef := aAxisRef[7],  iPersistentDataStorage := fbPersistentDataStorage, sName := 'Axis_07'),
		(AxisRef := aAxisRef[8],  iPersistentDataStorage := fbPersistentDataStorage, sName := 'Axis_08'),
		(AxisRef := aAxisRef[9],  iPersistentDataStorage := fbPersistentDataStorage, sName := 'Axis_09'),
		(AxisRef := aAxisRef[10], iPersistentDataStorage := fbPersistentDataStorage, sName := 'Axis_10'),
		(AxisRef := aAxisRef[11], iPersistentDataStorage := fbPersistentDataStorage, sName := 'Axis_11'),
		(AxisRef := aAxisRef[12], iPersistentDataStorage := fbPersistentDataStorage, sName := 'Axis_12'),
		(AxisRef := aAxisRef[13], iPersistentDataStorage := fbPersistentDataStorage, sName := 'Axis_13'),
		(AxisRef := aAxisRef[14], iPersistentDataStorage := fbPersistentDataStorage, sName := 'Axis_14'),
		(AxisRef := aAxisRef[15], iPersistentDataStorage := fbPersistentDataStorage, sName := 'Axis_15'),
		(AxisRef := aAxisRef[16], iPersistentDataStorage := fbPersistentDataStorage, sName := 'Axis_16'),
		(AxisRef := aAxisRef[17], iPersistentDataStorage := fbPersistentDataStorage, sName := 'Axis_17'),
		(AxisRef := aAxisRef[18], iPersistentDataStorage := fbPersistentDataStorage, sName := 'Axis_18'),
		(AxisRef := aAxisRef[19], iPersistentDataStorage := fbPersistentDataStorage, sName := 'Axis_19'),
		(AxisRef := aAxisRef[20], iPersistentDataStorage := fbPersistentDataStorage, sName := 'Axis_20'),
		(AxisRef := aAxisRef[21], iPersistentDataStorage := fbPersistentDataStorage, sName := 'Axis_21'),
		(AxisRef := aAxisRef[22], iPersistentDataStorage := fbPersistentDataStorage, sName := 'Axis_22'),
		(AxisRef := aAxisRef[23], iPersistentDataStorage := fbPersistentDataStorage, sName := 'Axis_23'),
		(AxisRef := aAxisRef[24], iPersistentDataStorage := fbPersistentDataStorage, sName := 'Axis_24'),
		(AxisRef := aAxisRef[25], iPersistentDataStorage := fbPersistentDataStorage, sName := 'Axis_25'),
		(AxisRef := aAxisRef[26], iPersistentDataStorage := fbPersistentDataStorage, sName := 'Axis_26'),
		(AxisRef := aAxisRef[27], iPersistentDataStorage := fbPersistentDataStorage, sName := 'Axis_27'),
		(AxisRef := aAxisRef[28], iPersistentDataStorage := fbPersistentDataStorage, sName := 'Axis_28'),
		(AxisRef := aAxisRef[29], iPersistentDataStorage := fbPersistentDataStorage, sName := 'Axis_29'),
		(AxisRef := aAxisRef[30], iPersistentDataStorage := fbPersistentDataStorage, sName := 'Axis_30'),
		(AxisRef := aAxisRef[31], iPersistentDataStorage := fbPersistentDataStorage, sName := 'Axis_31'),
		(AxisRef := aAxisRef[32], iPersistentDataStorage := fbPersistentDataStorage, sName := 'Axis_32'),
		(AxisRef := aAxisRef[33], iPersistentDataStorage := fbPersistentDataStorage, sName := 'Axis_33'),
		(AxisRef := aAxisRef[34], iPersistentDataStorage := fbPersistentDataStorage, sName := 'Axis_34'),
		(AxisRef := aAxisRef[35], iPersistentDataStorage := fbPersistentDataStorage, sName := 'Axis_35'),
		(AxisRef := aAxisRef[36], iPersistentDataStorage := fbPersistentDataStorage, sName := 'Axis_36'),
		(AxisRef := aAxisRef[37], iPersistentDataStorage := fbPersistentDataStorage, sName := 'Axis_37'),
		(AxisRef := aAxisRef[38], iPersistentDataStorage := fbPersistentDataStorage, sName := 'Axis_38'),
		(AxisRef := aAxisRef[39], iPersistentDataStorage := fbPersistentDataStorage, sName := 'Axis_39'),
		(AxisRef := aAxisRef[40], iPersistentDataStorage := fbPersistentDataStorage, sName := 'Axis_40'),
		(AxisRef := aAxisRef[41], iPersistentDataStorage := fbPersistentDataStorage, sName := 'Axis_41'),
		(AxisRef := aAxisRef[42], iPersistentDataStorage := fbPersistentDataStorage, sName := 'Axis_42'),
		(AxisRef := aAxisRef[43], iPersistentDataStorage := fbPersistentDataStorage, sName := 'Axis_43'),
		(AxisRef := aAxisRef[44], iPersistentDataStorage := fbPersistentDataStorage, sName := 'Axis_44'),
		(AxisRef := aAxisRef[45], iPersistentDataStorage := fbPersistentDataStorage, sName := 'Axis_45'),
		(AxisRef := aAxisRef[46], iPersistentDataStorage := fbPersistentDataStorage, sName := 'Axis_46'),
		(AxisRef := aAxisRef[47], iPersistentDataStorage := fbPersistentDataStorage, sName := 'Axis_47'),
		(AxisRef := aAxisRef[48], iPersistentDataStorage := fbPersistentDataStorage, sName := 'Axis_48'),
		(AxisRef := aAxisRef[49], iPersistentDataStorage := fbPersistentDataStorage, sName := 'Axis_49'),
		(AxisRef := aAxisRef[50], iPersistentDataStorage := fbPersistentDataStorage, sName := 'Axis_50')
	];

    {attribute 'pytmc' :='
        pv: @(PREFIX)INCR
        io: i
    '}
    stIncr: ST_PytmcTypes;
    {attribute 'pytmc' :='
        pv: @(PREFIX)SET
        io: io
    '}
    stSet: ST_PytmcTypes;

    timer: TON := (PT := T#2S);
    rand: DRAND;
    idx: UINT;
    mult: LREAL;
	nI : UINT;
END_VAR
VAR PERSISTENT
    {attribute 'pytmc' :='
        pv: @(PREFIX)PERS:PASS0
        io: io
		autosave_pass0: VAL
    '}
	afPersistentPass0: ARRAY[1..nInArray] OF LREAL;
    {attribute 'pytmc' :='
        pv: @(PREFIX)PERS:PASS1
        io: io
		autosave_pass1: VAL
    '}
	afPersistentPass1: ARRAY[1..nInArray] OF LREAL;
END_VAR


fbMotion01(stMotionStage:=M1);
fbMotion02(stMotionStage:=M2);

FOR nI := 1 TO nMotAbsAxes BY 1 DO
	fbMotionArr[nI]();
END_FOR

timer(
    IN:=NOT timer.Q
);

IF timer.Q THEN
	// Flip the boolean
	stIncr.bBool := NOT stIncr.bBool;

	// Increment the ints
	stIncr.iByte := stIncr.iByte + 1;
	stIncr.iSint := stIncr.iSint + 1;
	stIncr.iUsint := stIncr.iUsint + 1;
	stIncr.iWord := stIncr.iWord + 1;
	stIncr.iInt := stIncr.iInt + 1;
	stIncr.iUint := stIncr.iUint + 1;
	stIncr.iDword := stIncr.iDword + 1;
	stIncr.iDint := stIncr.iDint + 1;
	stIncr.iUdint := stIncr.iUdint + 1;

	// Multiply the floats randomly
	rand(Seed:=42);
	IF rand.Num < 0.5 THEN
		mult := rand.Num + 0.5;
	ELSE
		mult := rand.Num * 2;
	END_IF
	IF stIncr.fReal = 0 THEN
		stIncr.fReal := 1;
	ELSIF stIncr.fReal > 99999999.9999 THEN
		stIncr.fReal := 1;
	ELSE
		stIncr.fReal := LREAL_TO_REAL(stIncr.fReal * mult);
	END_IF
	IF stIncr.fLreal = 0 THEN
		stIncr.fLreal := 1;
	ELSIF stIncr.fLreal > 99999999.9999 THEN
		stIncr.fLreal := 1;
	ELSE
		stIncr.fLreal := stIncr.fLreal * mult;
	END_IF

	// To the next enum
	CASE stIncr.eEnum OF
		ENUM_Test.zero : stIncr.eEnum := Enum_test.one;
		ENUM_Test.one : stIncr.eEnum := Enum_test.two;
		ENUM_Test.two : stIncr.eEnum := Enum_test.three;
		ENUM_Test.three : stIncr.eEnum := Enum_test.four;
		ENUM_Test.four : stIncr.eEnum := Enum_test.five;
		ENUM_Test.five : stIncr.eEnum := Enum_test.six;
		ENUM_Test.six : stIncr.eEnum := Enum_test.seven;
		ENUM_Test.seven : stIncr.eEnum := Enum_test.zero;
	END_CASE

	// I guess we'll just do the letter a a lot
	IF LEN(stIncr.sString) > 39 THEN
		stIncr.sString := '';
	ELSE
		stIncr.sString := CONCAT(stIncr.sString, 'a');
	END_IF
	
	// I guess we'll just do the letter b a lot
	IF LEN(stIncr.sMaxString) > 254 THEN
		stIncr.sMaxString := '';
	ELSE
		stIncr.sMaxString := CONCAT(stIncr.sMaxString, 'b');
	END_IF

	F_UpdateArray(stIncr := stIncr);
END_IF

END_PROGRAM

// ---- POUs/F_UpdateArray.TcPOU

FUNCTION F_UpdateArray 
VAR_IN_OUT
	stIncr : ST_PytmcTypes;
END_VAR
VAR
	idx : UINT;
END_VAR


// Array, copy value to next and add one in first slot
FOR idx := 0 TO GVL.nPytmcTypesArrayLength - 1 DO
	stIncr.arrBool[GVL.nPytmcTypesArrayLength - idx] := stIncr.arrBool[GVL.nPytmcTypesArrayLength - 1 - idx];
END_FOR
stIncr.arrBool[0] := NOT stIncr.arrBool[0];

// pytmc cannot handle byte arrays we should fix that...
// FOR idx := 0 TO GVL.nPytmcTypesArrayLength - 1 DO
// 	stIncr.arrByte[GVL.nPytmcTypesArrayLength - idx] := stIncr.arrByte[GVL.nPytmcTypesArrayLength - 1 - idx];
// END_FOR
// stIncr.arrByte[0] := stIncr.arrByte[0] + 1;

// pytmc cannot handle sint arrays we should fix that...
// FOR idx := 0 TO GVL.nPytmcTypesArrayLength - 1 DO
// 	stIncr.arrSint[GVL.nPytmcTypesArrayLength - idx] := stIncr.arrSint[GVL.nPytmcTypesArrayLength - 1 - idx];
// END_FOR
// stIncr.arrSint[0] := stIncr.arrSint[0] + 1;

// pytmc cannot handle usint arrays we should fix that...
// FOR idx := 0 TO GVL.nPytmcTypesArrayLength - 1 DO
// 	stIncr.arrUsint[GVL.nPytmcTypesArrayLength - idx] := stIncr.arrUsint[GVL.nPytmcTypesArrayLength - 1 - idx];
// END_FOR
// stIncr.arrUsint[0] := stIncr.arrUsint[0] + 1;

// pytmc cannot handle word arrays we should fix that...
// FOR idx := 0 TO GVL.nPytmcTypesArrayLength - 1 DO
// 	stIncr.arrWord[GVL.nPytmcTypesArrayLength - idx] := stIncr.arrWord[GVL.nPytmcTypesArrayLength - 1 - idx];
// END_FOR
// stIncr.arrWord[0] := stIncr.arrWord[0] + 1;

FOR idx := 0 TO GVL.nPytmcTypesArrayLength - 1 DO
	stIncr.arrInt[GVL.nPytmcTypesArrayLength - idx] := stIncr.arrInt[GVL.nPytmcTypesArrayLength - 1 - idx];
END_FOR
stIncr.arrInt[0] := stIncr.arrInt[0] + 1;

// pytmc cannot handle uint arrays we should fix that...
// FOR idx := 0 TO GVL.nPytmcTypesArrayLength - 1 DO
// 	stIncr.arrUint[GVL.nPytmcTypesArrayLength - idx] := stIncr.arrUint[GVL.nPytmcTypesArrayLength - 1 - idx];
// END_FOR
// stIncr.arrUint[0] := stIncr.arrUint[0] + 1;

// pytmc cannot handle dword arrays we should fix that...
// FOR idx := 0 TO GVL.nPytmcTypesArrayLength - 1 DO
// 	stIncr.arrDword[GVL.nPytmcTypesArrayLength - idx] := stIncr.arrDword[GVL.nPytmcTypesArrayLength - 1 - idx];
// END_FOR
// stIncr.arrDword[0] := stIncr.arrDword[0] + 1;

FOR idx := 0 TO GVL.nPytmcTypesArrayLength - 1 DO
	stIncr.arrDint[GVL.nPytmcTypesArrayLength - idx] := stIncr.arrDint[GVL.nPytmcTypesArrayLength - 1 - idx];
END_FOR
stIncr.arrDint[0] := stIncr.arrDint[0] + 1;

// pytmc cannot handle udint arrays we should fix that...
// FOR idx := 0 TO GVL.nPytmcTypesArrayLength - 1 DO
// 	stIncr.arrUdint[GVL.nPytmcTypesArrayLength - idx] := stIncr.arrUdint[GVL.nPytmcTypesArrayLength - 1 - idx];
// END_FOR
// stIncr.arrUdint[0] := stIncr.arrUdint[0] + 1;

FOR idx := 0 TO GVL.nPytmcTypesArrayLength - 1 DO
	stIncr.arrReal[GVL.nPytmcTypesArrayLength - idx] := stIncr.arrReal[GVL.nPytmcTypesArrayLength - 1 - idx];
END_FOR
stIncr.arrReal[0] := stIncr.arrReal[0] + 1.0;

FOR idx := 0 TO GVL.nPytmcTypesArrayLength - 1 DO
	stIncr.arrLreal[GVL.nPytmcTypesArrayLength - idx] := stIncr.arrLreal[GVL.nPytmcTypesArrayLength - 1 - idx];
END_FOR
stIncr.arrLreal[0] := stIncr.arrLreal[0] + 1.0;

END_FUNCTION
